TYPE U_NCI_CTRL :
UNION

  stCtrl              : ARRAY[1..MAX_NCI_CH] OF ST_NCI_CTRL;

  byCtrl    AT %I*    : ARRAY[1..MAX_NCI_CH] OF
                        ARRAY[1..SIZEOF(ST_NCI_CTRL)] OF BYTE;
END_UNION
END_TYPE

(* stored: Version 1.1.0.1, ProductVersion 3.1.4026.13
   DUT U_NCI_CTRL: Id {62639e53-a363-4b03-95cb-c65461d36c94} *)
